// Mitsubishi GX Works2 project: dmddyd2   PLC: Q02/Q02H

PROGRAM MAIN
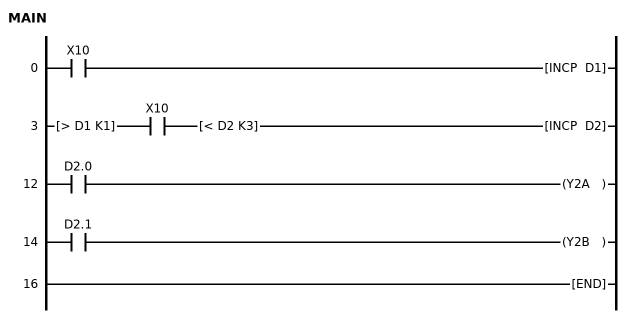
0     LD      X10
      INCP    D1
3     LD>     D1 K1
      AND     X10
      AND<    D2 K3
      INCP    D2
12    LD      D2.0
      OUT     Y2A
14    LD      D2.1
      OUT     Y2B
16    END
END_PROGRAM
